    CASE OP_Arr_OP160P[Output_Page_num] OF
    700: OLine6:= "O140_LK_TST1 _SEL4(Q700.5)        ";
    701: OLine6:= "O140_LK_TST2 _SEL3(Q701.5)        ";
    702: OLine6:= "O140_LK_TST3 _SEL2(Q702.5)        ";
    703: OLine6:= "O140_LK_TST4 _SEL1(Q703.5)        ";
    704: OLine6:= "O140_LK_TST5 _STRT(Q704.5)        ";
    705: OLine6:= "O140_LK_TST6 _RST(Q705.5)         ";
    706: OLine6:= "O140_LK_TST6 _SEL7(Q706.5)        ";
    707: OLine6:= "O160_SAMPLE_PART_DOR_OPN(Q707.5) ";
    708: OLine6:= "O10A_DRUM_RST(Q708.5)             ";
    709: OLine6:= "O160_SPARE_Q709_5(Q709.5)         ";
   1340: OLine6:= "O130_LH_TOOL_CHO_LOCK(Q1340.5)";
   1341: OLine6:= "O140_TOOL1_CHO_LOCK(Q1341.5)";
   1342: OLine6:= "O140_TOOL2_CHO_LOCK(Q1342.5)";
   1343: OLine6:= "O140_TOOL3_CHO_LOCK(Q1343.5)";
   1350: OLine6:= "O160_SLIDE_CYL_FWD(Q1350.5)";
   1351: OLine6:= "O160_RH_PALLET_LOCK_CYL_LOCK(Q1351.5)";
   1352: OLine6:= "O160_SPARE_Q1352_5(Q1352.5)";
   1353: OLine6:= "O160_SPARE_Q1353_5(Q1353.5)";
    ELSE
      OLine6:= " ";	
    END_CASE
       Out_Visibility_6:=TRUE;
	
    CASE OP_Arr_OP160P[Output_Page_num] OF
	700:  Out_Lamp6:=O140_LK_TST1_SEL4_Q700_5;
	701:  Out_Lamp6:=O140_LK_TST2_SEL3_Q701_5;
	702:  Out_Lamp6:=O140_LK_TST3_SEL2_Q702_5;
	703:  Out_Lamp6:=O140_LK_TST4_SEL1_Q703_5;
	704:  Out_Lamp6:=O140_LK_TST5_STRT_Q704_5;
	705:  Out_Lamp6:=O140_LK_TST6_RST_Q705_5;
	706:  Out_Lamp6:=O140_LK_TST6_SEL7_Q706_5;
	707:  Out_Lamp6:=O160_SAMPLE_PART_DOOR_OPN_Q707_5;
	708:  Out_Lamp6:=O10A_DRUM_RST_Q708_5;
	709:  Out_Lamp6:=O160_SPARE_Q709_5;
	1340: Out_Lamp6:=O130_LH_TOOL_CHO_LOCK_Q1340_5;
	1341: Out_Lamp6:=O140_TOOL1_CHO_LOCK_Q1341_5;
	1342: Out_Lamp6:=O140_TOOL2_CHO_LOCK_Q1342_5;
	1343: Out_Lamp6:=O140_TOOL3_CHO_LOCK_Q1343_5;
	1350: Out_Lamp6:=O160_SLIDE_CYL_FWD_Q1350_5;
	1351: Out_Lamp6:=O160_RH_PALLET_LOCK_CYL_LOCK_Q1351_5;
	1352: Out_Lamp6:=O160_SPARE_Q1352_5;
	1353: Out_Lamp6:=O160_SPARE_Q1353_5;
   ELSE           
       Out_Visibility_6:=FALSE;
   END_CASE 
       
    CASE OP_Arr_OP160P[Output_Page_num] OF
    700: OLine7:= "O140_LK_TST1 _SEL5(Q700.6)    ";
    701: OLine7:= "O140_LK_TST2 _SEL4(Q701.6)    ";
    702: OLine7:= "O140_LK_TST3 _SEL3(Q702.6)    ";
    703: OLine7:= "O140_LK_TST4 _SEL2(Q703.6)    ";
    704: OLine7:= "O140_LK_TST5 _SEL1(Q704.6)    ";
    705: OLine7:= "O140_LK_TST6 _STRT(Q705.6)    ";
    706: OLine7:= "O150_VISN_LGHT_ON(Q706.6)     ";
    707: OLine7:= "O160_REJ_BIN_DOR_OPN(Q707.6) ";
    708: OLine7:= "O10A_DRUM_EXT_SPEED(Q708.6)   ";
    709: OLine7:= "O160_SPARE_Q709_6(Q709.6)     ";
   1340: OLine7:= "O130_RH_TOOL_CHO_UNLOCK(Q1340.6)";
   1341: OLine7:= "O140_WIPE1_CYL_REV(Q1341.6)";
   1342: OLine7:= "O140_WIPE2_CYL_REV(Q1342.6)";
   1343: OLine7:= "O140_WIPE3_CYL_REV(Q1343.6)";
   1350: OLine7:= "O160_SPARE_Q1350_6(Q1350.6)";
   1351: OLine7:= "O160_SPARE_Q1351_6(Q1351.6)";
   1352: OLine7:= "O160_SPARE_Q1352_6(Q1352.6)";
   1353: OLine7:= "O160_SPARE_Q1353_6(Q1353.6)";
    ELSE
      OLine7:= " ";	
    END_CASE
       Out_Visibility_7:=TRUE;
	
   CASE OP_Arr_OP160P[Output_Page_num] OF
	700:  Out_Lamp7:=O140_LK_TST1_SEL5_Q700_6;
	701:  Out_Lamp7:=O140_LK_TST2_SEL4_Q701_6;
	702:  Out_Lamp7:=O140_LK_TST3_SEL3_Q702_6;
	703:  Out_Lamp7:=O140_LK_TST4_SEL2_Q703_6;
	704:  Out_Lamp7:=O140_LK_TST5_SEL1_Q704_6;
	705:  Out_Lamp7:=O140_LK_TST6_STRT_Q705_6;
	706:  Out_Lamp7:=O150_VISN_LGHT_ON_Q706_6;
	707:  Out_Lamp7:=O160_REJ_BIN_DOOR_OPN_Q707_6;
	708:  Out_Lamp7:=O10A_DRUM_EXT_SPEED_Q708_6;
	709:  Out_Lamp7:=O160_SPARE_Q709_6;
	1340: Out_Lamp7:=O130_RH_TOOL_CHO_UNLOCK_Q1340_6;
	1341: Out_Lamp7:=O140_WIPE1_CYL_REV_Q1341_6;
	1342: Out_Lamp7:=O140_WIPE2_CYL_REV_Q1342_6;
	1343: Out_Lamp7:=O140_WIPE3_CYL_REV_Q1343_6;
	1350: Out_Lamp7:=O160_SPARE_Q1350_6;
	1351: Out_Lamp7:=O160_SPARE_Q1351_6;
	1352: Out_Lamp7:=O160_SPARE_Q1352_6;
	1353: Out_Lamp7:=O160_SPARE_Q1353_6;
   ELSE
       Out_Visibility_7:=FALSE;
   END_CASE 
    
    CASE OP_Arr_OP160P[Output_Page_num] OF
    700: OLine8:= "O140_LK_TST1_SEL6(Q700.7)";
    701: OLine8:= "O140_LK_TST2_SEL5(Q701.7)";
    702: OLine8:= "O140_LK_TST3_SEL4(Q702.7)";
    703: OLine8:= "O140_LK_TST4_SEL3(Q703.7)";
    704: OLine8:= "O140_LK_TST5_SEL2(Q704.7)";
    705: OLine8:= "O140_LK_TST6_SEL1(Q705.7)";
    706: OLine8:= "O150_BARLIGHT_OP1(Q706.7) ";
    707: OLine8:= "O160_SPARE(Q707.7)        ";
    708: OLine8:= "O160_SPARE_Q708_7(Q708.7) ";
    709: OLine8:= "O160_SPARE_Q709_7(Q709.7) ";
   1340: OLine8:= "O130_RH_TOOL_CHO_LOCK(Q1340.7)";
   1341: OLine8:= "O140_WIPE1_CYL_FWD(Q1341.7)";
   1342: OLine8:= "O140_WIPE2_CYL_FWD(Q1342.7)";
   1343: OLine8:= "O140_WIPE3_CYL_FWD(Q1343.7)";
   1350: OLine8:= "O160_SPARE_Q1350_7(Q1350.7)";
   1351: OLine8:= "O160_SPARE_Q1351_7(Q1351.7)";
   1352: OLine8:= "O160_SPARE_Q1352_7(Q1352.7)";
   1353: OLine8:= "O160_SPARE_Q1353_7(Q1353.7)";
    ELSE
      OLine8:= " ";	
    END_CASE	
       Out_Visibility_8:=TRUE;
   
   CASE OP_Arr_OP160P[Output_Page_num] OF
	700:  Out_Lamp8:=O140_LK_TST1_SEL6_Q700_7;
	701:  Out_Lamp8:=O140_LK_TST2_SEL5_Q701_7;
	702:  Out_Lamp8:=O140_LK_TST3_SEL4_Q702_7;
	703:  Out_Lamp8:=O140_LK_TST4_SEL3_Q703_7;
	704:  Out_Lamp8:=O140_LK_TST5_SEL2_Q704_7;
	705:  Out_Lamp8:=O140_LK_TST6_SEL1_Q705_7;
	706:  Out_Lamp8:=O150_BARLIGHT_OP1_Q706_7;
	707:  Out_Lamp8:=O160_SPARE_Q707_7;
	708:  Out_Lamp8:=O160_SPARE_Q708_7;
	709:  Out_Lamp8:=O160_SPARE_Q709_7;
	1340: Out_Lamp8:=O130_RH_TOOL_CHO_LOCK_Q1340_7;
	1341: Out_Lamp8:=O140_WIPE1_CYL_FWD_Q1341_7;
	1342: Out_Lamp8:=O140_WIPE2_CYL_FWD_Q1342_7;
	1343: Out_Lamp8:=O140_WIPE3_CYL_FWD_Q1343_7;
	1350: Out_Lamp8:=O160_SPARE_Q1350_7;
	1351: Out_Lamp8:=O160_SPARE_Q1351_7;
	1352: Out_Lamp8:=O160_SPARE_Q1352_7;
	1353: Out_Lamp8:=O160_SPARE_Q1353_7;
   ELSE
       Out_Visibility_8:=FALSE;	
   END_CASE 
  
 4: CASE IP_Arr_OP10A[Input_Page_num] OF
      100:Line1:="I10A_HPR_UNIT_ALRM(I100.0)    ";
      101:Line1:="I10A_HPR_DOOR_SELCTN(I101.0)  ";
      102:Line1:="I10A_LNR_TRK1_CHO_MOD1(I102.0)";
      103:Line1:="I10A_SPARE_I103_0(I103.0)     ";
      ELSE
      	Line1:= " ";
      END_CASE
      
      CASE IP_Arr_OP10A[Input_Page_num] OF
      100:Line2:="I10A_SPARE_I100.1(I100.1)      ";
      101:Line2:="I10A_SPARE_I101.1(I101.1)      ";
      102:Line2:="I10A_LNR_TRK1_CHO_MOD2(I102.1) ";
      103:Line2:="I10A_SPARE_I103_1(I103.1)      ";
      ELSE
      	Line2 := " ";
      END_CASE
      
      CASE IP_Arr_OP10A[Input_Page_num] OF
      100:Line3:="I10A_HPR_LOW_LVL_SEN(I100.2)   ";
      101:Line3:="I10A_BDY_BOWL_LOW_LVL(I101.2)  ";
      102:Line3:="I10A_LNR_TRK2_CHO_MOD1(I102.2) ";
      103:Line3:="I10A_SPARE_I103_2(I103.2)      ";
      ELSE
      	Line3 := " ";
      END_CASE
      
      CASE IP_Arr_OP10A[Input_Page_num] OF
      100:Line4:="I10A_HPR_SOL_DOOR_SW_FB(I100.3)";
      101:Line4:="I10A_BDY_BWL_RUN(I101.3)       ";
      102:Line4:="I10A_LNR_TRK2_CHO_MOD2(I102.3) ";
      103:Line4:="I10A_SPARE_I103_3(I103.3)      ";
      ELSE
      	Line4 := " ";
      END_CASE
      
      CASE IP_Arr_OP10A[Input_Page_num] OF
      100:Line5:="I10A_HPR_OFF_ON(I100.4)";
      101:Line5:="I10A_BDY_LNR1_RUN(I101.4)";
      102:Line5:="I10A_SPARE_I102_4(I102.4)";
      103:Line5:="I10A_SPARE_I103_4(I103.4)";
      ELSE
      	Line5:= " ";
      END_CASE
      
      CASE IP_Arr_OP10A[Input_Page_num] OF
      100:Line6:="I10A_BDY_BOWL_OFF_ON(I100.5)  ";
      101:Line6:="I10A_BDY_LNR2_RUN(I101.5)     ";
      102:Line6:="I10A_SPARE_I102_5(I102.5)";
      103:Line6:="I10A_SPARE_I103_5(I103.5)     ";
      ELSE
      	Line6 := " ";
      END_CASE
      
      CASE IP_Arr_OP10A[Input_Page_num] OF
      100:Line7:="I10A_BDY_LNR1_OFF_ON(I100.6)     ";
      101:Line7:="I10A_BDY_LNR_FEED1_OVRFLW(I101.6)";
      102:Line7:="I10A_LH_BDY_CONT_FB(I102.6)      ";
      103:Line7:="I10A_SPARE_I103_6(I103.6)        ";
      ELSE
      	Line7 := " ";
      END_CASE
      
      CASE IP_Arr_OP10A[Input_Page_num] OF
      100:Line8:="I10A_BDY_LNR2_OFF_ON(I100.7)     ";
      101:Line8:="I10A_BDY_LNR_FEED2_OVRFLW(I101.7)";
      102:Line8:="I10A_RH_BDY_CONT_FB(I102.7)      ";
      103:Line8:="I10A_SPARE_I103_7(I103.7)        ";
      ELSE
      	Line8 := " ";
      END_CASE
	 	Visibility_1:=TRUE;
   
   CASE IP_Arr_OP10A[Input_Page_num] OF
	100: Lamp1:=I10A_HPR_UNIT_ALRM_I100_0 ;
	101: Lamp1:=I10A_HPR_DOOR_SELCTN_I101_0 ;
	102: Lamp1:=I10A_LNR_TRK1_CHO_MOD1_I102_0 ;
	103: Lamp1:=I10A_SPARE_I103_0;
   ELSE
       Visibility_1:=FALSE;	
   END_CASE
   
   Visibility_2:=TRUE;
   
   CASE IP_Arr_OP10A[Input_Page_num] OF
	100: Lamp2:=I10A_SPARE_I100_1 ;
	101: Lamp2:=I10A_SPARE_I101_1;
	102: Lamp2:=I10A_LNR_TRK1_CHO_MOD2_I102_1 ;
	103: Lamp2:=I10A_SPARE_I103_1;
   ELSE
       Visibility_2:=FALSE;	
   END_CASE
   
   
    Visibility_3:=TRUE;
   
   CASE IP_Arr_OP10A[Input_Page_num] OF
	100: Lamp3:=I10A_HPR_LOW_LVL_SEN_I100_2 ;
	101: Lamp3:=I10A_BDY_BOWL_LOW_LVL_I101_2 ;
	102: Lamp3:=I10A_LNR_TRK2_CHO_MOD1_I102_2 ;
	103: Lamp3:=I10A_SPARE_I103_2;
   ELSE
       Visibility_3:=FALSE;	
   END_CASE
   
   
    Visibility_4:=TRUE;
   
   CASE IP_Arr_OP10A[Input_Page_num] OF
	100: Lamp4:=I10A_HPR_SOL_DOOR_SW_FB_I100_3 ;
	101: Lamp4:=I10A_BDY_BWL_RUN_I101_3 ;
	102: Lamp4:=I10A_LNR_TRK2_CHO_MOD2_I102_3 ;
	103: Lamp4:=I10A_SPARE_I103_3;
   ELSE
       Visibility_4:=FALSE;	
   END_CASE
   
   
    
    Visibility_5:=TRUE;
   
   CASE IP_Arr_OP10A[Input_Page_num] OF
	100: Lamp5:=I10A_HPR_OFF_ON_I100_4 ;
	101: Lamp5:=I10A_BDY_LNR1_RUN_I101_4 ;
	102: Lamp5:=I10A_SPARE_I102_4 ;
	103: Lamp5:=I10A_SPARE_I103_4;
   ELSE
       Visibility_5:=FALSE;	
   END_CASE
   
    
    Visibility_6:=TRUE;
   
   CASE IP_Arr_OP10A[Input_Page_num] OF
	100: Lamp6:=I10A_BDY_BOWL_OFF_ON_I100_5 ;
	101: Lamp6:=I10A_BDY_LNR2_RUN_I101_5 ;
	102: Lamp6:=I10A_SPARE_I102_5 ;
	103: Lamp6:=I10A_SPARE_I103_5;
   ELSE
       Visibility_6:=FALSE;	
   END_CASE
   
   
      
    Visibility_7:=TRUE;
   
   CASE IP_Arr_OP10A[Input_Page_num] OF
	100: Lamp7:=I10A_BDY_LNR1_OFF_ON_I100_6 ;
	101: Lamp7:=I10A_BDY_LNR_FEED1_OVRFLW_I101_6 ;
	102: Lamp7:=I10A_LH_BDY_CONT_FB_I102_6;
	103: Lamp7:=I10A_SPARE_I103_6;
   ELSE
       Visibility_7:=FALSE;	
   END_CASE


 	Visibility_8:=TRUE;
   
   CASE IP_Arr_OP10A[Input_Page_num] OF
	100: Lamp8:=I10A_BDY_LNR2_OFF_ON_I100_7 ;
	101: Lamp8:=I10A_BDY_LNR_FEED2_OVRFLW_I101_7 ;
	102: Lamp8:=I10A_RH_BDY_CONT_FB_I102_7 ;
	103: Lamp8:=I10A_SPARE_I103_7;
   ELSE
       Visibility_8:=FALSE;	
   END_CASE

	
	 CASE OP_Arr_OP10A[Output_Page_num] OF
     100:OLine1:="O10A_HPR_MTR_FWD(Q100.0)  ";
     101:OLine1:="O10A_BDY_BOWL_ON(Q101.0)  ";
     102:OLine1:="O10A_SPARE_Q102_0(Q102.0) ";
     103:OLine1:="O10A_SPARE_Q103_0(Q103.0) ";
     ELSE
     	OLine1:= " ";
     END_CASE
     
     CASE OP_Arr_OP10A[Output_Page_num] OF
     100:OLine2:="O10A_HPR_RST(Q100.1)         ";
     101:OLine2:="O10A_BDY_LNR_FEED1_ON(Q101.1)";
     102:OLine2:="O10A_SPARE_Q102_1(Q102.1)    ";
     103:OLine2:="O10A_SPARE_Q103_1(Q103.1)    ";
     ELSE
     	OLine2:= " ";
     END_CASE
     
     CASE OP_Arr_OP10A[Output_Page_num] OF
     100:OLine3:="O10A_EXT_SPEED(Q100.2)       ";
     101:OLine3:="O10A_BDY_LNR_FEED2_ON(Q101.2)";
     102:OLine3:="O10A_SPARE_Q102_2(Q102.2)    ";
     103:OLine3:="O10A_SPARE_Q103_2(Q103.2)    ";
     ELSE
     	OLine3:= " ";
     END_CASE
     
     CASE OP_Arr_OP10A[Output_Page_num] OF
     100:OLine4:="O10A_SPARE_Q100.3(Q100.3)      ";
     101:OLine4:="O10A_BDY_LNR1_AIR_PURGE(Q101.3)";
     102:OLine4:="O10A_SPARE_Q102_3(Q102.3)      ";
     103:OLine4:="O10A_SPARE_Q103_3(Q103.3)      ";
     ELSE
     	OLine4:= " ";
     END_CASE
     
     CASE OP_Arr_OP10A[Output_Page_num] OF
     100:OLine5:="O10A_HPR_DOOR_SELCTN_IND(Q100.4)";
   //101:OLine5:="O10A_BDY_LNR2_AIRPURGE(Q101.4)";
     102:OLine5:="O10A_SPARE_Q102_4(Q102.4)";
     103:OLine5:="O10A_SPARE_Q103_4(Q103.4)";
     ELSE
     	OLine5:= " ";
     END_CASE
     
     CASE OP_Arr_OP10A[Output_Page_num] OF
     100:OLine6:="O10A_HPR_TWR_LMP_RED(Q100.5)";
     101:OLine6:="O10A_HPR_DOOR_OPN(Q101.5)   ";
     102:OLine6:="O10A_SPARE_Q102_5(Q102.5)   ";
     103:OLine6:="O10A_SPARE_Q103_5(Q103.5)   ";
     ELSE
     	OLine6:= " ";
     END_CASE
     
     CASE OP_Arr_OP10A[Output_Page_num] OF
     100:OLine7:="O10A_HPR_TWR_LMP_GREEN(Q100.6)";
     101:OLine7:="O10A_SPARE_Q101_6(Q101.6)     ";
     102:OLine7:="O10A_SPARE_Q102_6(Q102.6)     ";
     103:OLine7:="O10A_SPARE_Q103_6(Q103.6)     ";
     ELSE
     	OLine7:= " ";
     END_CASE
     
     CASE OP_Arr_OP10A[Output_Page_num] OF
     100:OLine8:="O10A_SPARE_Q100_7(Q100.7)";
     101:OLine8:="O10A_SPARE_Q101_7(Q101.7)";
     102:OLine8:="O10A_SPARE_Q102_7(Q102.7)";
     103:OLine8:="O10A_SPARE_Q103_7(Q103.7)";
     ELSE
     	OLine8:= " ";
     END_CASE
	  Out_Visibility_1:=TRUE;

    CASE OP_Arr_OP10A[Output_Page_num] OF
	100:  Out_Lamp1:=O10A_HPR_MTR_FWD_Q100_0;
	101:  Out_Lamp1:=O10A_BDY_BOWL_ON_Q101_0;
	102:  Out_Lamp1:=O10A_SPARE_Q102_0;
	103:  Out_Lamp1:=O10A_SPARE_Q103_0;
   ELSE
       Out_Visibility_1:=FALSE;	
   END_CASE
   
    Out_Visibility_2:=TRUE;
   
   CASE OP_Arr_OP10A[Output_Page_num] OF
	100:  Out_Lamp2:=O10A_HPR_RST_Q100_1;
	101:  Out_Lamp2:=O10A_BDY_LNR_FEED1_ON_Q101_1;
	102:  Out_Lamp2:=O10A_SPARE_Q102_1;
	103:  Out_Lamp2:=O10A_SPARE_Q103_1;
   ELSE
       Out_Visibility_2:=FALSE;	
   END_CASE 
   
    Out_Visibility_3:=TRUE;
	
   CASE OP_Arr_OP10A[Output_Page_num] OF
	100:  Out_Lamp3:=O10A_EXT_SPEED_Q100_2; 
	101:  Out_Lamp3:=O10A_BDY_LNR_FEED2_ON_Q101_2; 
	102:  Out_Lamp3:=O10A_SPARE_Q102_2; 
	103:  Out_Lamp3:=O10A_SPARE_Q103_2; 
   ELSE
       Out_Visibility_3:=FALSE;
   END_CASE 
   
    Out_Visibility_4:=TRUE;
   
   CASE OP_Arr_OP10A[Output_Page_num] OF
	100:  Out_Lamp4:=O10A_SPARE_Q100_3; 
	101:  Out_Lamp4:=O10A_BDY_LNR1_AIR_PURGE_Q101_3; 
	102:  Out_Lamp4:=O10A_SPARE_Q102_3; 
	103:  Out_Lamp4:=O10A_SPARE_Q103_3;  
   ELSE
       Out_Visibility_4:=FALSE;
   END_CASE 
   
    Out_Visibility_5:=TRUE;
	
    CASE OP_Arr_OP10A[Output_Page_num] OF
	100:  Out_Lamp5:=O10A_HPR_DOOR_SELCTN_IND_Q100_4; 
	//101:  Out_Lamp5:=O10A_BDY_LNR2_AIR_PURGE_Q101_4; 
	102:  Out_Lamp5:=O10A_SPARE_Q102_4; 
	103:  Out_Lamp5:=O10A_SPARE_Q103_4; 	 
   ELSE
       Out_Visibility_5:=FALSE;
   END_CASE 
   
    Out_Visibility_6:=TRUE;
	
   CASE OP_Arr_OP10A[Output_Page_num] OF
	100:  Out_Lamp6:=O10A_HPR_TWR_LMP_RED_Q100_5; 
	101:  Out_Lamp6:=O10A_HPR_DOOR_OPN_Q101_5; 
	102:  Out_Lamp6:=O10A_SPARE_Q102_5; 
	103:  Out_Lamp6:=O10A_SPARE_Q103_5; 
   ELSE           
       Out_Visibility_6:=FALSE;
   END_CASE 
    
	Out_Visibility_7:=TRUE;
	
   CASE OP_Arr_OP10A[Output_Page_num] OF
	100:  Out_Lamp7:=O10A_HPR_TWR_LMP_GREEN_Q100_6; 
	101:  Out_Lamp7:=O10A_SPARE_Q101_6; 
	102:  Out_Lamp7:=O10A_SPARE_Q102_6; 
	103:  Out_Lamp7:=O10A_SPARE_Q103_6;  
   ELSE 
       Out_Visibility_7:=FALSE;
   END_CASE 
   
    Out_Visibility_8:=TRUE;
   
   CASE OP_Arr_OP10A[Output_Page_num] OF
	100:  Out_Lamp8:=O10A_SPARE_Q100_7;  
	101:  Out_Lamp8:=O10A_SPARE_Q101_7;  
	102:  Out_Lamp8:=O10A_SPARE_Q102_7;  
	103:  Out_Lamp8:=O10A_SPARE_Q103_7;   
   ELSE
       Out_Visibility_8:=FALSE;	
   END_CASE
	 
 5: CASE IP_Arr_OP10B[Input_Page_num] OF
    200: Line1:= "I10B_HPR_UNIT_ALRM(I200.0)     ";
    201: Line1:= "I10B_HPR_DOOR_SELCTN(I201.0)   ";
    202: Line1:= "I10B_LNR_TRK1_CHO_MOD1(I202.0) ";
    203: Line1:= "I10B_SPARE_I203_0(I203.0)      ";
    ELSE
    	Line1 := " ";
    END_CASE
    
    CASE IP_Arr_OP10B[Input_Page_num] OF
    200: Line2:= "I10B_SPARE_I200_1(I200.1)     ";
    201: Line2:= "I10B_SPARE_I201_1(I201.1)     ";
    202: Line2:= "I10B_LNR_TRK1_CHO_MOD2(I202.1)";
    203: Line2:= "I10B_SPARE_I203_1(I203.1)     ";
    ELSE
    	Line2 := " ";
    END_CASE
    
    CASE IP_Arr_OP10B[Input_Page_num] OF
    200: Line3:= "I10B_HPR_LOW_LVL_SEN(I200.2)   ";
    201: Line3:= "I10B_BDY_BOWL_LOW_LVL(I201.2)  ";
    202: Line3:= "I10B_LNR_TRK2_CHO_MOD1(I202.2) ";
    203: Line3:= "I10B_SPARE_I203_2(I203.2)      ";
    ELSE
    	Line3 := " ";
    END_CASE
    
    CASE IP_Arr_OP10B[Input_Page_num] OF
    200: Line4:= "I10B_HPR_SOL_DOOR_SW_FB(I200.3)";
    201: Line4:= "I10B_BDY_BWL_RUN(I201.3)       ";
    202: Line4:= "I10B_LNR_TRK2_CHO_MOD2(I202.3) ";
    203: Line4:= "I10B_SPARE_I203_3(I203.3)      ";
    ELSE
    	Line4 := " ";
    END_CASE
    
    CASE IP_Arr_OP10B[Input_Page_num] OF
    200: Line5:= "I10B_HPR_OFF_ON(I200.4)       ";
    201: Line5:= "I10B_BDY_LNR1_RUN(I201.4)     ";
    202: Line5:= "I10B_SPARE_I202_4(I202.4)";
    203: Line5:= "I10B_SPARE_I203_4(I203.4)     ";
    ELSE
    	Line5 := " ";
    END_CASE
    
    CASE IP_Arr_OP10B[Input_Page_num] OF
    200: Line6:= "I10B_BDY_BOWL_OFF_ON(I200.5)   ";
    201: Line6:= "I10B_BDY_LNR2_RUN(I201.5)      ";
    202: Line6:= "I10B_SPARE_I202_5(I202.5) ";
    203: Line6:= "I10B_SPARE_I203_5(I203.5)      ";
    ELSE
    	Line6 := " ";
    END_CASE
    
    CASE IP_Arr_OP10B[Input_Page_num] OF
    200: Line7:= "I10B_BDY_LNR1_OFF_ON(I200.6)      ";
    201: Line7:= "I10B_BDY_LNR_FEED1_OVRFLW(I201.6) ";
    202: Line7:= "I10B_SPARE_I202_6(I202.6)         ";
    203: Line7:= "I10B_SPARE_I203_6(I203.6)         ";
    ELSE
    	Line7 := " ";
    END_CASE
    
    CASE IP_Arr_OP10B[Input_Page_num] OF
    200: Line8:= "I10B_BDY_LNR2_OFF_ON(I200.7)     ";
    201: Line8:= "I10B_BDY_LNR_FEED2_OVRFLW(I201.7)";
    202: Line8:= "I10B_SPARE_I202_7(I202.7)        ";
    203: Line8:= "I10B_SPARE_I203_7(I203.7)        ";
    ELSE
    	Line8 := " ";
    END_CASE
	  Visibility_1:=TRUE;
   
   CASE IP_Arr_OP10B[Input_Page_num] OF
	200: Lamp1:=I10B_HPR_UNIT_ALRM_I200_0 ;
	201: Lamp1:=I10B_HPR_DOOR_SELCTN_I201_0 ;
	202: Lamp1:=I10B_LNR_TRK1_CHO_MOD1_I202_0 ;
	203: Lamp1:=I10B_SPARE_I203_0;
   ELSE
       Visibility_1:=FALSE;	
   END_CASE
   
   
   Visibility_2:=TRUE;
   
   CASE IP_Arr_OP10B[Input_Page_num] OF
	200: Lamp2:=I10B_SPARE_I200_1 ;
	201: Lamp2:=I10B_SPARE_I201_1 ;
	202: Lamp2:=I10B_LNR_TRK1_CHO_MOD2_I202_1 ;
	203: Lamp2:=I10B_SPARE_I203_1;
   ELSE
       Visibility_2:=FALSE;	
   END_CASE
   
   
    Visibility_3:=TRUE;
   
   CASE IP_Arr_OP10B[Input_Page_num] OF
	200: Lamp3:=I10B_HPR_LOW_LVL_SEN_I200_2 ;
	201: Lamp3:=I10B_BDY_BOWL_LOW_LVL_I201_2 ; 
	202: Lamp3:=I10B_LNR_TRK2_CHO_MOD1_I202_2 ;
	203: Lamp3:=I10B_SPARE_I203_2 ;
   ELSE
       Visibility_3:=FALSE;	
   END_CASE
   
   
    Visibility_4:=TRUE;
   
   CASE IP_Arr_OP10B[Input_Page_num] OF
	200: Lamp4:=I10B_HPR_SOL_DOOR_SW_FB_I200_3 ;
	201: Lamp4:=I10B_BDY_BWL_RUN_I201_3 ; 
	202: Lamp4:=I10B_LNR_TRK2_CHO_MOD2_I202_3 ;
	203: Lamp4:=I10B_SPARE_I203_3 ;
   ELSE
       Visibility_4:=FALSE;	
   END_CASE
   
   
    Visibility_5:=TRUE;
   
   CASE IP_Arr_OP10B[Input_Page_num] OF
	200: Lamp5:=I10B_HPR_OFF_ON_I200_4 ;
	201: Lamp5:=I10B_BDY_LNR1_RUN_I201_4 ;
	202: Lamp5:=I10B_SPARE_I202_4 ;
	203: Lamp5:=I10B_SPARE_I203_4;
   ELSE
       Visibility_5:=FALSE;	
   END_CASE
   
    
    Visibility_6:=TRUE;
   
   CASE IP_Arr_OP10B[Input_Page_num] OF
	200: Lamp6:=I10B_BDY_BOWL_OFF_ON_I200_5 ;
	201: Lamp6:=I10B_BDY_LNR2_RUN_I201_5 ;
	202: Lamp6:=I10B_SPARE_I202_5 ;
	203: Lamp6:=I10B_SPARE_I203_5 ;
   ELSE
       Visibility_6:=FALSE;	
   END_CASE
   
      
    Visibility_7:=TRUE;
   
   CASE IP_Arr_OP10B[Input_Page_num] OF
	200: Lamp7:=I10B_BDY_LNR1_OFF_ON_I200_6 ;
	201: Lamp7:=I10B_BDY_LNR_FEED1_OVRFLW_I201_6 ;
	202: Lamp7:=I10B_SPARE_I202_6 ;
	203: Lamp7:=I10B_SPARE_I203_6;
   ELSE
       Visibility_7:=FALSE;	
   END_CASE


    Visibility_8:=TRUE;
   
   CASE IP_Arr_OP10B[Input_Page_num] OF
	200: Lamp8:=I10B_BDY_LNR2_OFF_ON_I200_7 ;
	201: Lamp8:=I10B_BDY_LNR_FEED2_OVRFLW_I201_7 ;
	202: Lamp8:=I10B_SPARE_I202_7 ;
	203: Lamp8:=I10B_SPARE_I203_7;
   ELSE
       Visibility_8:=FALSE;	
   END_CASE


  CASE OP_Arr_OP10B_JB[Output_Page_num] OF	
  200: OLine1:= " O10B_HPR_MTR_FWD(Q200.0) ";
  201: OLine1:= " O10B_BDY_BOWL_ON(Q201.0) ";
  202: OLine1:= " O10B_SPARE_Q202_0(Q202.0)";
  203: OLine1:= " O10B_SPARE_Q203_0(Q203.0)";
  ELSE
      OLine1 := " ";
  END_CASE
  
  CASE OP_Arr_OP10B_JB[Output_Page_num] OF
  200: OLine2:= "O10B_HPR_RST(Q200.1)         ";
  201: OLine2:= "O10B_BDY_LNR_FEED1_ON(Q201.1)";
  202: OLine2:= "O10B_SPARE_Q202_1(Q202.1)    ";
  203: OLine2:= "O10B_SPARE_Q203_1(Q203.1)    ";
  ELSE
    OLine2 := " ";
  END_CASE
  
  CASE OP_Arr_OP10B_JB[Output_Page_num] OF
  200: OLine3:= "O10B_EXT_SPEED(Q200.2)       ";
  201: OLine3:= "O10B_BDY_LNR_FEED2_ON(Q201.2)";
  202: OLine3:= "O10B_SPARE_Q202_2(Q202.2)    ";
  203: OLine3:= "O10B_SPARE_Q2032_(Q203.2)    ";
  ELSE
    OLine3 := " ";
  END_CASE
  
  CASE OP_Arr_OP10B_JB[Output_Page_num] OF
  200: OLine4:= "O10B_SPARE_Q200.3(Q200.3)      ";
  201: OLine4:= "O10B_BDY_LNR1_AIR_PURGE(Q201.3)";
  202: OLine4:= "O10B_SPARE_Q202_3(Q202.3)      ";
  203: OLine4:= "O10B_SPARE_Q203_3(Q203.3)      ";
  ELSE
    OLine4 := " ";
  END_CASE
  
  CASE OP_Arr_OP10B_JB[Output_Page_num] OF
  200: OLine5:= "O10B_HPR_DOOR_SELCTN_IND(Q200.4)";
  //201: OLine5:= "O10B_BDY_LNR2_AIR_PURGE(Q201.4) ";
  202: OLine5:= "O10B_SPARE_Q202_4(Q202.4)       ";
  203: OLine5:= "O10B_SPARE_Q203_4(Q203.4)       ";
  ELSE
     OLine5 := " ";
  END_CASE
  
  CASE OP_Arr_OP10B_JB[Output_Page_num] OF
  200: OLine6:= "O10B_HPR_TWR_LMP_RED(Q200.5)";
  201: OLine6:= "O10B_HPR_DOOR_OPN(Q201.5)   ";
  202: OLine6:= "O10B_SPARE_Q202_5(Q202.5)   ";
  203: OLine6:= "O10B_SPARE_Q203_5(Q203.5)   ";
  ELSE
     OLine6 := " ";
  END_CASE
  
  CASE OP_Arr_OP10B_JB[Output_Page_num] OF
  200: OLine7:= "O10B_HPR_TWR_LMP_GREEN(Q200.6)";
  201: OLine7:= "O10B_SPARE_Q201_6(Q201.6)     ";
  202: OLine7:= "O10B_SPARE_Q202_6(Q202.6)     ";
  203: OLine7:= "O10B_SPARE_Q203_6(Q203.6)     ";
  ELSE
      OLine7 := " ";
  END_CASE
  
  CASE OP_Arr_OP10B_JB[Output_Page_num] OF	 
  200: OLine8:= "O10B_SPARE_Q200_7(Q200.7)";
  201: OLine8:= "O10B_SPARE_Q201_7(Q201.7)";
  202: OLine8:= "O10B_SPARE_Q202_7(Q202.7)";
  203: OLine8:= "O10B_SPARE_Q203_7(Q203.7)";
  ELSE
      OLine8 := " ";
  END_CASE	

    Out_Visibility_1:=TRUE;

   CASE OP_Arr_OP10B_JB[Output_Page_num] OF
	200:  Out_Lamp1:=O10B_HPR_MTR_FWD_Q200_0;
	201:  Out_Lamp1:=O10B_BDY_BOWL_ON_Q201_0;
	202:  Out_Lamp1:=O10B_SPARE_Q202_0;
	203:  Out_Lamp1:=O10B_SPARE_Q203_0;
   ELSE
       Out_Visibility_1:=FALSE;	
   END_CASE
   
    Out_Visibility_2:=TRUE;
   
   CASE OP_Arr_OP10B_JB[Output_Page_num] OF
	200:  Out_Lamp2:=O10B_HPR_RST_Q200_1;
	201:  Out_Lamp2:=O10B_BDY_LNR_FEED1_ON_Q201_1;
	202:  Out_Lamp2:=O10B_SPARE_Q202_1;
	203:  Out_Lamp2:=O10B_SPARE_Q203_1;
   ELSE
       Out_Visibility_2:=FALSE;	
   END_CASE 
   
    Out_Visibility_3:=TRUE;
	
   CASE OP_Arr_OP10B_JB[Output_Page_num] OF
	200:  Out_Lamp3:=O10B_EXT_SPEED_Q200_2; 
	201:  Out_Lamp3:=O10B_BDY_LNR_FEED2_ON_Q201_2; 
	202:  Out_Lamp3:=O10B_SPARE_Q202_2; 
	203:  Out_Lamp3:=O10B_SPARE_Q203_2; 
   ELSE
       Out_Visibility_3:=FALSE;
   END_CASE 
   
    Out_Visibility_4:=TRUE;
   
   CASE OP_Arr_OP10B_JB[Output_Page_num] OF
	200:  Out_Lamp4:=O10B_SPARE_Q200_3; 
	201:  Out_Lamp4:=O10B_BDY_LNR1_AIR_PURGE_Q201_3; 
	202:  Out_Lamp4:=O10B_SPARE_Q202_3; 
	203:  Out_Lamp4:=O10B_SPARE_Q203_3;  
   ELSE
       Out_Visibility_4:=FALSE;
   END_CASE 
   
    Out_Visibility_5:=TRUE;
	
    CASE OP_Arr_OP10B_JB[Output_Page_num] OF
	200:  Out_Lamp5:=O10B_HPR_DOOR_SELCTN_IND_Q200_4; 
	201:  Out_Lamp5:=O10B_BDY_LNR2_AIR_PURGE_Q201_4 ; 
	202:  Out_Lamp5:=O10B_SPARE_Q202_4; 
	203:  Out_Lamp5:=O10B_SPARE_Q203_4; 	 
   ELSE
       Out_Visibility_5:=FALSE;
   END_CASE 
   
    Out_Visibility_6:=TRUE;
	
   CASE OP_Arr_OP10B_JB[Output_Page_num] OF
	200:  Out_Lamp6:=O10B_HPR_TWR_LMP_RED_Q200_5; 
	201:  Out_Lamp6:=O10B_HPR_DOOR_OPN_Q201_5; 
	202:  Out_Lamp6:=O10B_SPARE_Q202_5; 
	203:  Out_Lamp6:=O10B_SPARE_Q203_5; 
   ELSE           
       Out_Visibility_6:=FALSE;
   END_CASE 
    
	Out_Visibility_7:=TRUE;
	
   CASE OP_Arr_OP10B_JB[Output_Page_num] OF
	200:  Out_Lamp7:=O10B_HPR_TWR_LMP_GREEN_Q200_6; 
	201:  Out_Lamp7:=O10B_SPARE_Q201_6; 
	202:  Out_Lamp7:=O10B_SPARE_Q202_6; 
	203:  Out_Lamp7:=O10B_SPARE_Q203_6;  
   ELSE 
       Out_Visibility_7:=FALSE;
   END_CASE 
   
    Out_Visibility_8:=TRUE;
   
   CASE OP_Arr_OP10B_JB[Output_Page_num] OF
	200:  Out_Lamp8:=O10B_SPARE_Q200_7;  
	201:  Out_Lamp8:=O10B_SPARE_Q201_7;  
	202:  Out_Lamp8:=O10B_SPARE_Q202_7;  
	203:  Out_Lamp8:=O10B_SPARE_Q203_7;   
   ELSE
       Out_Visibility_8:=FALSE;	
   END_CASE 
 6: CASE IP_Arr_OP90JB[Input_Page_num] OF
    500: Line1:=" I90_SPARE_I500_0(I500.0)       ";
    501: Line1:=" I90_CONV1_FWD(I501.0)          ";
    502: Line1:=" I90_CONV1_TRK3_CHO_MOD2(I502.0)";
    503: Line1:=" I90_CONV2_REV(I503.0)          ";
    504: Line1:=" I90_CONV2_TRK3_CHO_MOD1(I504.0)";
    505: Line1:=" I90_SPARE_I505_0(I505.0)       ";
    else
     Line1:=" ";
    end_case 
    
    CASE IP_Arr_OP90JB[Input_Page_num] OF
    500: Line2:="I90_HPR1_LOW_LVL_FB(I500.1)        ";
    501: Line2:="I90_VBF1_CONV1_TRK1_OVERFLW(I501.1)";
    502: Line2:="I90_SPARE_I502_1(I502.1)           ";
    503: Line2:="I90_CONV2_FWD(I503.1)              ";
    504: Line2:="I90_CONV2_TRK3_CHO_MOD2(I504.1)    ";
    505: Line2:="I90_SPARE_I505_1(I505.1)           ";
    else
     Line2:=" ";
    end_case 
    
    CASE IP_Arr_OP90JB[Input_Page_num] OF
    500: Line3:="I90_HPR1_SOL_DOOR_SW_FB(I500.2)    ";
    501: Line3:="I90_VBF1_CONV1_TRK2_OVERFLW(I501.2)";
    502: Line3:="I90_HPR2_LOW_LVL_FB(I502.2)        ";
    503: Line3:="I90_VBF1_CONV2_TRK1_OVERFLW(I503.2)";
    504: Line3:="I90_VBF1_CONV_TRK_OVERFLW_2(I504.2)";
    505: Line3:="I90_SPARE_I505_2(I505.2)           ";
    else
     Line3:=" ";
    end_case 
    
    CASE IP_Arr_OP90JB[Input_Page_num] OF
    500: Line4:="I90_BOWL1_RDY(I500.3)              ";
    501: Line4:="I90_CONV1_TRK1_CHO_MOD1(I501.3)    ";
    502: Line4:="I90_HPR2_SOL_DOOR_SW_FB(I502.3)    ";
    503: Line4:="I90_VBF1_CONV2_TRK2_OVERFLW(I503.3)";
    504: Line4:="I90_VBF2_CONV_TRK_OVERFLW_2(I504.3)";
    505: Line4:="I90_SPARE_I505_3(I505.3)           ";
    else
     Line4:=" ";
    end_case 
    
    CASE IP_Arr_OP90JB[Input_Page_num] OF
    500: Line5:="I90_BOWL1_LOW_LVL(I500.4)      ";
    501: Line5:="I90_CONV1_TRK1_CHO_MOD2(I501.4)";
    502: Line5:="I90_BOWL2_RDY(I502.4)          ";
    503: Line5:="I90_CONV2_TRK1_CHO_MOD1(I503.4)";
    504: Line5:="I90_SPARE_I504_4(I504.4)       ";
    505: Line5:="I90_SPARE_I505_4(I505.4)       ";
    else
     Line5:=" ";
    end_case 
    
    CASE IP_Arr_OP90JB[Input_Page_num] OF
    500: Line6:="I90_BOWL1_OFF_ON(I500.5)        ";
    501: Line6:="I90_CONV1_TRK2_CHO_MOD1(I501.5) ";
    502: Line6:="I90_BOWL2_LOW_LVL(I502.5)       ";
    503: Line6:="I90_CONV2_TRK1_CHO_MOD2(I503.5) ";
    504: Line6:="I90_SPARE_I504_5(I504.5)        ";
    505: Line6:="I90_SPARE_I505_5(I505.5)        ";
    else
     Line6:=" ";
    end_case 
    
    CASE IP_Arr_OP90JB[Input_Page_num] OF
    500: Line7:="I90_HPR1_OFF_ON(I500.6)        ";
    501: Line7:="I90_CONV1_TRK2_CHO_MOD2(I501.6)";
    502: Line7:="I90_BOWL2_OFF_ON(I502.6)       ";
    503: Line7:="I90_CONV2_TRK2_CHO_MOD1(I503.6)";
    504: Line7:="I90_SPARE_I504_6(I504.6)       ";
    505: Line7:="I90_SPARE_I505_6(I505.6)       ";
    else
     Line7:=" ";
    end_case 
    
    CASE IP_Arr_OP90JB[Input_Page_num] OF
    500: Line8:="I90_CONV1_REV(I500.7)           ";
    501: Line8:="I90_CONV1_TRK3_CHO_MOD1(I501.7) ";
    502: Line8:="I90_HPR2_OFF_ON(I502.7)         ";
    503: Line8:="I90_CONV2_TRK2_CHO_MOD2(I503.7) ";
    504: Line8:="I90_SPARE_I504_7(I504.7)        ";
    505: Line8:="I90_SPARE_I505_7(I505.7)        ";
    else
     Line8:=" ";
    END_CASE 
	
  Visibility_1:=TRUE;
   
   CASE IP_Arr_OP90JB[Input_Page_num] OF
	500: Lamp1:=I90_SPARE_I500_0 ;
	501: Lamp1:=I90_CONV1_FWDI501_0 ;
	502: Lamp1:=I90_CONV1_TRK3_CHO_MOD2I502_0 ;
	503: Lamp1:=I90_CONV2_REVI503_0;
	504: Lamp1:=I90_CONV2_TRK3_CHO_MOD1I504_0 ;
	505: Lamp1:=I90_SPARE_I505_0 ;
   ELSE
       Visibility_1:=FALSE;	
   END_CASE
   
   
   Visibility_2:=TRUE;
   
   CASE IP_Arr_OP90JB[Input_Page_num] OF
	500: Lamp2:=I90_HPR1_LOW_LVL_FBI500_1 ;
	501: Lamp2:=I90_VBF1_CONV1_TRK1_OVERFLWI501_1 ;
	502: Lamp2:=I90_SPARE_I502_1 ;
	503: Lamp2:=I90_CONV2_FWDI503_1;
	504: Lamp2:=I90_CONV2_TRK3_CHO_MOD2I504_1 ;
	505: Lamp2:=I90_SPARE_I505_1 ;
   ELSE
       Visibility_2:=FALSE;	
   END_CASE
   
   
    Visibility_3:=TRUE;
   
   CASE IP_Arr_OP90JB[Input_Page_num] OF
	500: Lamp3:=I90_HPR1_SOL_DOOR_SW_FBI500_2 ;
	501: Lamp3:=I90_VBF1_CONV1_TRK2_OVERFLWI501_2 ;
	502: Lamp3:=I90_HPR2_LOW_LVL_FBI502_2 ;
	503: Lamp3:=I90_VBF1_CONV2_TRK1_OVERFLWI503_2;
	504: Lamp3:=I90_VBF1_CONV_TRK_OVERFLW_2I504_2 ;
	505: Lamp3:=I90_SPARE_I505_2 ;
   ELSE
       Visibility_3:=FALSE;	
   END_CASE
   
   
    Visibility_4:=TRUE;
   
   CASE IP_Arr_OP90JB[Input_Page_num] OF
	500: Lamp4:=I90_BOWL1_RDYI500_3 ;
	501: Lamp4:=I90_CONV1_TRK1_CHO_MOD1I501_3 ;
	502: Lamp4:=I90_HPR2_SOL_DOOR_SW_FBI502_3 ;
	503: Lamp4:=I90_VBF1_CONV2_TRK2_OVERFLWI503_3;
	504: Lamp4:=I90_VBF2_CONV_TRK_OVERFLW_2I504_3 ;
	505: Lamp4:=I90_SPARE_I505_3 ;
   ELSE
       Visibility_4:=FALSE;	
   END_CASE
   
   
    Visibility_5:=TRUE;
   
   CASE IP_Arr_OP90JB[Input_Page_num] OF
	500: Lamp5:=I90_BOWL1_LOW_LVLI500_4 ;
	501: Lamp5:=I90_CONV1_TRK1_CHO_MOD2I501_4 ;
	502: Lamp5:=I90_BOWL2_RDYI502_4 ;
	503: Lamp5:=I90_CONV2_TRK1_CHO_MOD1I503_4;
	504: Lamp5:=I90_SPARE_I504_4 ;
	505: Lamp5:=I90_SPARE_I505_4 ;
   ELSE
       Visibility_5:=FALSE;	
   END_CASE
   
   
    Visibility_6:=TRUE;
   
   CASE IP_Arr_OP90JB[Input_Page_num] OF
	500: Lamp6:=I90_BOWL1_OFF_ONI500_5 ;
	501: Lamp6:=I90_CONV1_TRK2_CHO_MOD1I501_5 ;
	502: Lamp6:=I90_BOWL2_LOW_LVLI502_5 ;
	503: Lamp6:=I90_CONV2_TRK1_CHO_MOD2I503_5;
	504: Lamp6:=I90_SPARE_I504_5 ;
	505: Lamp6:=I90_SPARE_I505_5 ;
   ELSE
       Visibility_6:=FALSE;	
   END_CASE
   
   
    Visibility_7:=TRUE;
   
   CASE IP_Arr_OP90JB[Input_Page_num] OF
	500: Lamp7:=I90_HPR1_OFF_ONI500_6 ;
	501: Lamp7:=I90_CONV1_TRK2_CHO_MOD2I501_6 ;
	502: Lamp7:=I90_BOWL2_OFF_ONI502_6 ;
	503: Lamp7:=I90_CONV2_TRK2_CHO_MOD1I503_6;
	504: Lamp7:=I90_SPARE_I504_6 ;
	505: Lamp7:=I90_SPARE_I505_6 ;
   ELSE
       Visibility_7:=FALSE;	
   END_CASE
   
   
    Visibility_8:=TRUE;
   
   CASE IP_Arr_OP90JB[Input_Page_num] OF
	500: Lamp8:=I90_CONV1_REVI500_7 ;
	501: Lamp8:=I90_CONV1_TRK3_CHO_MOD1I501_7 ;
	502: Lamp8:=I90_HPR2_OFF_ONI502_7 ;
	503: Lamp8:=I90_CONV2_TRK2_CHO_MOD2I503_7;
	504: Lamp8:=I90_SPARE_I504_7 ;
	505: Lamp8:=I90_SPARE_I505_7 ;
   ELSE
       Visibility_8:=FALSE;	
   END_CASE
	
    CASE OP_Arr_OP90[Output_Page_num] OF
    500: OLine1:=" O90_HPR1_ENABLE(Q500.0)  ";
    501: OLine1:=" O90_HPR2_ENABLE(Q501.0)  ";
    502: OLine1:=" O90_SPARE_Q502_0(Q502.0) ";
    503: OLine1:=" O90_SPARE_Q503_0(Q503.0) ";
    else
     OLine1:=" ";
    end_case 
    
    CASE OP_Arr_OP90[Output_Page_num] OF
    500: OLine2:="O90_BOWL1_ENABLE(Q500.1)";
    501: OLine2:="O90_BOWL2_ENABLE(Q501.1)";
    502: OLine2:="O90_SPARE_Q502_1(Q502.1)";
    503: OLine2:="O90_SPARE_Q503_1(Q503.1)";
    else
     OLine2:=" ";
    end_case 
    
    CASE OP_Arr_OP90[Output_Page_num] OF
    500: OLine3:="O90_HPR1_TWR_LMP_RED(Q500.2)";
    501: OLine3:="O90_HPR2_TWR_LMP_RED(Q501.2)";
    502: OLine3:="O90_SPARE_Q502_2(Q502.2)    ";
    503: OLine3:="O90_SPARE_Q503_2(Q503.2)    ";
    else
     OLine3:=" ";
    end_case 
    
    CASE OP_Arr_OP90[Output_Page_num] OF
    500: OLine4:="O90_HPR1_TWR_LMP_GREEN(Q500.3)";
    501: OLine4:="O90_HPR2_TWR_LMP_GREEN(Q501.3)";
    502: OLine4:="O90_SPARE_Q502_3(Q502.3)      ";
    503: OLine4:="O90_SPARE_Q503_3(Q503.3)      ";
    else
     OLine4:=" ";
    end_case 
    
    CASE OP_Arr_OP90[Output_Page_num] OF
    500: OLine5:="O90_BOWL1_AIR_PURGE1(Q500.4)";
    501: OLine5:="O90_BOWL2_AIR_PURGE1(Q501.4)";
    502: OLine5:="O90_SPARE_Q502_4(Q502.4)    ";
    503: OLine5:="O90_SPARE_Q503_4(Q503.4)    ";
    else
     OLine5:=" ";
    end_case 
    
    CASE OP_Arr_OP90[Output_Page_num] OF
    500: OLine6:="O90_BOWL1_AIR_PURGE2(Q500.5)";
    501: OLine6:="O90_BOWL2_AIR_PURGE2(Q501.5)";
    502: OLine6:="O90_SPARE_Q502_5(Q502.5)    ";
    503: OLine6:="O90_SPARE_Q503_5(Q503.5)    ";
    else
     OLine6:=" ";
    end_case 
    
    CASE OP_Arr_OP90[Output_Page_num] OF
    500: OLine7:="O90_HPR1_DOOR_OPN(Q500.6)";
    501: OLine7:="O90_HPR2_DOOR_OPN(Q501.6)";
    502: OLine7:="O90_SPARE_Q502_6(Q502.6) ";
    503: OLine7:="O90_SPARE_Q503_6(Q503.6) ";
    else
     OLine7:=" ";
    end_case 
    
    CASE OP_Arr_OP90[Output_Page_num] OF
    500: OLine8:="O90_SPARE_Q500_7(Q500.7)";
    501: OLine8:="O90_SPARE_Q501_7(Q501.7)";
    502: OLine8:="O90_SPARE_Q502_7(Q502.7)";
    503: OLine8:="O90_SPARE_Q503_7(Q503.7)";
    else
     OLine8:=" ";
    END_CASE 
    Out_Visibility_1:=TRUE;
    CASE OP_Arr_OP90[Output_Page_num] OF
	500:  Out_Lamp1:=O90_HPR1_ENABLEQ500_0;
	501:  Out_Lamp1:=O90_HPR2_ENABLEQ501_0;
	502:  Out_Lamp1:=O90_SPARE_Q502_0;
	503:  Out_Lamp1:=O90_SPARE_Q503_0;
    ELSE
       Out_Visibility_1:=FALSE;	
    END_CASE
   
    Out_Visibility_2:=TRUE;
   
    CASE OP_Arr_OP90[Output_Page_num] OF
	500:  Out_Lamp2:=O90_BOWL1_ENABLEQ500_1;
	501:  Out_Lamp2:=O90_BOWL2_ENABLEQ501_1;
	502:  Out_Lamp2:=O90_SPARE_Q502_1;
	503:  Out_Lamp2:=O90_SPARE_Q503_1;
    ELSE
       Out_Visibility_2:=FALSE;	
    END_CASE 
   
    Out_Visibility_3:=TRUE;
	
    CASE OP_Arr_OP90[Output_Page_num] OF
	500:  Out_Lamp3:=O90_HPR1_TWR_LMP_REDQ500_2; 
	501:  Out_Lamp3:=O90_HPR2_TWR_LMP_REDQ501_2; 
	502:  Out_Lamp3:=O90_SPARE_Q502_2; 
	503:  Out_Lamp3:=O90_SPARE_Q503_2; 
    ELSE
       Out_Visibility_3:=FALSE;
    END_CASE 
   
    Out_Visibility_4:=TRUE;
   
    CASE OP_Arr_OP90[Output_Page_num] OF
	500:  Out_Lamp4:=O90_HPR1_TWR_LMP_GREENQ500_3; 
	501:  Out_Lamp4:=O90_HPR2_TWR_LMP_GREENQ501_3; 
	502:  Out_Lamp4:=O90_SPARE_Q502_3; 
	503:  Out_Lamp4:=O90_SPARE_Q503_3;  
    ELSE
       Out_Visibility_4:=FALSE;
    END_CASE 
   
    Out_Visibility_5:=TRUE;
	
    CASE OP_Arr_OP90[Output_Page_num] OF
	500:  Out_Lamp5:=O90_BOWL1_AIR_PURGE1Q500_4; 
	501:  Out_Lamp5:=O90_BOWL2_AIR_PURGE1Q501_4; 
	502:  Out_Lamp5:=O90_SPARE_Q502_4; 
	503:  Out_Lamp5:=O90_SPARE_Q503_4; 
   ELSE
       Out_Visibility_5:=FALSE;
   END_CASE 
   
    Out_Visibility_6:=TRUE;
	
   CASE OP_Arr_OP90[Output_Page_num] OF
	500:  Out_Lamp6:=O90_BOWL1_AIR_PURGE2Q500_5; 
	501:  Out_Lamp6:=O90_BOWL2_AIR_PURGE2Q501_5; 
	502:  Out_Lamp6:=O90_SPARE_Q502_5; 
	503:  Out_Lamp6:=O90_SPARE_Q503_5; 
   ELSE           
       Out_Visibility_6:=FALSE;
   END_CASE 
    
	Out_Visibility_7:=TRUE;
	
   CASE OP_Arr_OP90[Output_Page_num] OF
	500:  Out_Lamp7:=O90_HPR1_DOOR_OPNQ500_6; 
	501:  Out_Lamp7:=O90_HPR2_DOOR_OPNQ501_6; 
	502:  Out_Lamp7:=O90_SPARE_Q502_6; 
	503:  Out_Lamp7:=O90_SPARE_Q503_6;  
   ELSE 
       Out_Visibility_7:=FALSE;
   END_CASE 
   
    Out_Visibility_8:=TRUE;
   
   CASE OP_Arr_OP90[Output_Page_num] OF
	500:  Out_Lamp8:=O90_SPARE_Q500_7;  
	501:  Out_Lamp8:=O90_SPARE_Q501_7;  
	502:  Out_Lamp8:=O90_SPARE_Q502_7;  
	503:  Out_Lamp8:=O90_SPARE_Q503_7;   
   ELSE
       Out_Visibility_8:=FALSE;	
   END_CASE
 7:	CASE IP_Arr_OP120_JB[Input_Page_num] OF
    600: Line1:="I120_SPARE_600_0(I600.0)        ";
    601: Line1:="I120_CONV_FWD(I601.0)           ";
    602: Line1:="I120_CONV_TRK3_CHO_MOD2(I602.0) ";
    603: Line1:="I120_SPARE_I603_0(I603.0)       ";
    else
     Line1:=" ";
    end_case 
     
    CASE IP_Arr_OP120_JB[Input_Page_num] OF
    600: Line2:="I120_HPR_LOW_LVL_FB(I600.1)       ";
    601: Line2:="I120_VBF_CONV_TRK1_OVERFLW(I601.1)";
    602: Line2:="I120_VBF_CONV_TRK_OVERFLW2(I602.1)   ";
    603: Line2:="I120_SPARE_I603_1(I603.1)         ";
    else
     Line2:=" ";
    end_case 
     
    CASE IP_Arr_OP120_JB[Input_Page_num] OF
    600: Line3:="I120_HPR_SOL_DOOR_SW_FB(I600.2)   ";
    601: Line3:="I120_VBF_CONV_TRK2_OVERFLW(I601.2)";
    602: Line3:="I120_SPARE_I602_2(I602.2)         ";
    603: Line3:="I120_SPARE_I603_2(I603.2)         ";
    else
     Line3:=" ";
    end_case 
     
    CASE IP_Arr_OP120_JB[Input_Page_num] OF
    600: Line4:="I120_BOWL_RDY(I600.3)          ";
    601: Line4:="I120_CONV_TRK1_CHO_MOD1(I601.3)";
    602: Line4:="I120_SPARE_I602_3(I602.3)      ";
    603: Line4:="I120_SPARE_I603_3(I603.3)      ";
    else
     Line4:=" ";
    end_case 
     
    CASE IP_Arr_OP120_JB[Input_Page_num] OF
    600: Line5:="I120_BOWL_LOW_LVL(I600.4)      ";
    601: Line5:="I120_CONV_TRK1_CHO_MOD2(I601.4)";
    602: Line5:="I120_SPARE_I602_4(I602.4)      ";
    603: Line5:="I120_SPARE_I603_4(I603.4)      ";
    else
     Line5:=" ";
    end_case 
     
    CASE IP_Arr_OP120_JB[Input_Page_num] OF
    600: Line6:="I120_BOWL_OFF_ON(I600.5)       ";
    601: Line6:="I120_CONV_TRK2_CHO_MOD1(I601.5)";
    602: Line6:="I120_SPARE_I602_5(I602.5)      ";
    603: Line6:="I120_SPARE_I603_5(I603.5)      ";
    else
     Line6:=" ";
    end_case 
     
    CASE IP_Arr_OP120_JB[Input_Page_num] OF
    600: Line7:="I120_HPR_OFF_ON(I600.6)        ";
    601: Line7:="I120_CONV_TRK2_CHO_MOD2(I601.6)";
    602: Line7:="I120_SPARE_I602_6(I602.6)      ";
    603: Line7:="I120_SPARE_I603_6(I603.6)      ";
    else
     Line7:=" ";
    end_case 
     
    CASE IP_Arr_OP120_JB[Input_Page_num] OF
    600: Line8:="I120_CONV_REV(I600.7)           ";
    601: Line8:="I120_CONV_TRK3_CHO_MOD1(I601.7) ";
    602: Line8:="I120_SPARE_I602_7(I602.7)       ";
    603: Line8:="I120_SPARE_I603_7(I603.7)       ";
    else
     Line8:=" ";
    END_CASE 
	Visibility_1:=TRUE;
   
   CASE IP_Arr_OP120_JB[Input_Page_num] OF
	600: Lamp1:=I120_SPARE_600_0I600_0 ;
	601: Lamp1:=I120_CONV_FWDI601_0 ;
	602: Lamp1:=I120_CONV_TRK3_CHO_MOD2I602_0 ;
	603: Lamp1:=I120_SPARE_I603_0;
   ELSE
       Visibility_1:=FALSE;	
   END_CASE
   
   
   Visibility_2:=TRUE;
   
   CASE IP_Arr_OP120_JB[Input_Page_num] OF
	600: Lamp2:=I120_HPR_LOW_LVL_FBI600_1 ;
	601: Lamp2:=I120_VBF_CONV_TRK1_OVERFLWI601_1 ;
	602: Lamp2:=I120_VBF_CONV_TRK_OVERFLW2I602_1 ;
	603: Lamp2:=I120_SPARE_I603_1;
   ELSE
       Visibility_2:=FALSE;	
   END_CASE
   
   
    Visibility_3:=TRUE;
   
   CASE IP_Arr_OP120_JB[Input_Page_num] OF
	600: Lamp3:=I120_HPR_SOL_DOOR_SW_FBI600_2 ;
	601: Lamp3:=I120_VBF_CONV_TRK2_OVERFLWI601_2 ;
	602: Lamp3:=I120_SPARE_I602_2 ;
	603: Lamp3:=I120_SPARE_I603_2;
   ELSE
       Visibility_3:=FALSE;	
   END_CASE

    Visibility_4:=TRUE;
   
   CASE IP_Arr_OP120_JB[Input_Page_num] OF
	600: Lamp4:=I120_BOWL_RDYI600_3 ;
	601: Lamp4:=I120_CONV_TRK1_CHO_MOD1I601_3 ;
	602: Lamp4:=I120_SPARE_I602_3 ;
	603: Lamp4:=I120_SPARE_I603_3;
   ELSE
       Visibility_4:=FALSE;	
   END_CASE
   
   
    Visibility_5:=TRUE;
   
   CASE IP_Arr_OP120_JB[Input_Page_num] OF
	600: Lamp5:=I120_BOWL_LOW_LVLI600_4 ;
	601: Lamp5:=I120_CONV_TRK1_CHO_MOD2I601_4 ;
	602: Lamp5:=I120_SPARE_I602_4 ;
	603: Lamp5:=I120_SPARE_I603_4;
   ELSE
       Visibility_5:=FALSE;	
   END_CASE
   
   
    Visibility_6:=TRUE;
   
   CASE IP_Arr_OP120_JB[Input_Page_num] OF
	600: Lamp6:=I120_BOWL_OFF_ONI600_5 ;
	601: Lamp6:=I120_CONV_TRK2_CHO_MOD1I601_5 ;
	602: Lamp6:=I120_SPARE_I602_5 ;
	603: Lamp6:=I120_SPARE_I603_5;
   ELSE
       Visibility_6:=FALSE;	
   END_CASE
   
   
    Visibility_7:=TRUE;
   
   CASE IP_Arr_OP120_JB[Input_Page_num] OF
	600: Lamp7:=I120_HPR_OFF_ONI600_6 ;
	601: Lamp7:=I120_CONV_TRK2_CHO_MOD2I601_6 ;
	602: Lamp7:=I120_SPARE_I602_6 ;
	603: Lamp7:=I120_SPARE_I603_6;
   ELSE
       Visibility_7:=FALSE;	
   END_CASE
   
   
    Visibility_8:=TRUE;
   
   CASE IP_Arr_OP120_JB[Input_Page_num] OF
	600: Lamp8:=I120_CONV_REVI600_7 ;
	601: Lamp8:=I120_CONV_TRK3_CHO_MOD1I601_7 ;
	602: Lamp8:=I120_SPARE_I602_7 ;
	603: Lamp8:=I120_SPARE_I603_7;
   ELSE
       Visibility_8:=FALSE;	
   END_CASE
    
    CASE OP_Arr_OP120[Output_Page_num] OF
    600: OLine1:="O120_HPR_ENABLE(Q600.0)   ";
    601: OLine1:="O120_SPARE_Q601_0(Q601.0) ";
    602: OLine1:="O120_SPARE_Q602_0(Q602.0) ";
    603: OLine1:="O120_SPARE_Q603_0(Q603.0) ";
    else
     OLine1:=" ";
    end_case 
    
    CASE OP_Arr_OP120[Output_Page_num] OF
    600: OLine2:="O120_BOWL_ENABLE(Q600.1) ";
    601: OLine2:="O120_SPARE_Q601_1(Q601.1)";
    602: OLine2:="O120_SPARE_Q602_1(Q602.1)";
    603: OLine2:="O120_SPARE_Q603_1(Q603.1)";
    else
     OLine2:=" ";
    end_case 
    
    CASE OP_Arr_OP120[Output_Page_num] OF
    600: OLine3:="O120_HPR_TWR_LMP_RED(Q600.2)";
    601: OLine3:="O120_SPARE_Q601_2(Q601.2)   ";
    602: OLine3:="O120_SPARE_Q602_2(Q602.2)   ";
    603: OLine3:="O120_SPARE_Q603_2(Q603.2)   ";
    else
     OLine3:=" ";
    end_case 
    
    CASE OP_Arr_OP120[Output_Page_num] OF
    600: OLine4:="O120_HPR_TWR_LMP_GREEN(Q600.3)";
    601: OLine4:="O120_SPARE_Q601.3(Q601.3)     ";
    602: OLine4:="O120_SPARE_Q602.3(Q602.3)     ";
    603: OLine4:="O120_SPARE_Q603.3(Q603.3)     ";
    else
     OLine4:=" ";
    end_case 
    
    CASE OP_Arr_OP120[Output_Page_num] OF
    600: OLine5:="O120_BOWL_AIR_PURGE1(Q600.4)";
    601: OLine5:="O120_SPARE_Q601_4(Q601.4)   ";
    602: OLine5:="O120_SPARE_Q602_4(Q602.4)   ";
    603: OLine5:="O120_SPARE_Q603_4(Q603.4)   ";
    else
     OLine5:=" ";
    end_case 
    
    CASE OP_Arr_OP120[Output_Page_num] OF
    600: OLine6:="O120_BOWL_AIR_PURGE2(Q600.5)";
    601: OLine6:="O120_SPARE_Q601_5(Q601.5)   ";
    602: OLine6:="O120_SPARE_Q602_5(Q602.5)   ";
    603: OLine6:="O120_SPARE_Q603_5(Q603.5)   ";
    else
     OLine6:=" ";
    end_case 
    
    CASE OP_Arr_OP120[Output_Page_num] OF
    600: OLine7:="O120_HPR_DOOR_OPN(Q600.6)";
    601: OLine7:="O120_SPARE_Q601_6(Q601.6)";
    602: OLine7:="O120_SPARE_Q602_6(Q602.6)";
    603: OLine7:="O120_SPARE_Q603_6(Q603.6)";
    else
     OLine7:=" ";
    end_case 
    
    CASE OP_Arr_OP120[Output_Page_num] OF
    600: OLine8:="O120_SPARE_Q600_7(Q600.7)";
    601: OLine8:="O120_SPARE_Q601_7(Q601.7)";
    602: OLine8:="O120_SPARE_Q602_7(Q602.7)";
    603: OLine8:="O120_SPARE_Q603_7(Q603.7)";
    else
     OLine8:=" ";
    END_CASE 
	   Out_Visibility_1:=TRUE;
   
   CASE OP_Arr_OP120[Output_Page_num] OF
	600:  Out_Lamp1:=O120_HPR_ENABLEQ600_0;
	601:  Out_Lamp1:=O120_SPARE_Q601_0;
	602:  Out_Lamp1:=O120_SPARE_Q602_0;
	603:  Out_Lamp1:=O120_SPARE_Q603_0;
   ELSE
       Out_Visibility_1:=FALSE;	
   END_CASE
   
    Out_Visibility_2:=TRUE;
   
   CASE OP_Arr_OP120[Output_Page_num] OF
	600:  Out_Lamp2:=O120_BOWL_ENABLEQ600_1;
	601:  Out_Lamp2:=O120_SPARE_Q601_1;
	602:  Out_Lamp2:=O120_SPARE_Q602_1;
	603:  Out_Lamp2:=O120_SPARE_Q603_1;
   ELSE
       Out_Visibility_2:=FALSE;	
   END_CASE 
   
    Out_Visibility_3:=TRUE;
	
   CASE OP_Arr_OP10A[Output_Page_num] OF
	600:  Out_Lamp3:=O120_HPR_TWR_LMP_REDQ600_2; 
	601:  Out_Lamp3:=O120_SPARE_Q601_2; 
	602:  Out_Lamp3:=O120_SPARE_Q602_2; 
	603:  Out_Lamp3:=O120_SPARE_Q603_2; 
   ELSE
       Out_Visibility_3:=FALSE;
   END_CASE 
   
    Out_Visibility_4:=TRUE;
   
   CASE OP_Arr_OP120[Output_Page_num] OF
	700:  Out_Lamp4:=O120_HPR_TWR_LMP_GREENQ600_3; 
	701:  Out_Lamp4:=O120_SPARE_Q601_3; 
	702:  Out_Lamp4:=O120_SPARE_Q602_3; 
	703:  Out_Lamp4:=O120_SPARE_Q603_3; 
   ELSE
       Out_Visibility_4:=FALSE;
   END_CASE 
   
    Out_Visibility_5:=TRUE;
	
    CASE OP_Arr_OP120[Output_Page_num] OF
	600:  Out_Lamp5:=O120_BOWL_AIR_PURGE1Q600_4; 
	601:  Out_Lamp5:=O120_SPARE_Q601_4; 
	602:  Out_Lamp5:=O120_SPARE_Q602_4; 
	603:  Out_Lamp5:=O120_SPARE_Q603_4; 
   ELSE
       Out_Visibility_5:=FALSE;
   END_CASE 
   
    Out_Visibility_6:=TRUE;
	
   CASE OP_Arr_OP120[Output_Page_num] OF
	600:  Out_Lamp6:=O120_BOWL_AIR_PURGE2Q600_5; 
	601:  Out_Lamp6:=O120_SPARE_Q601_5; 
	602:  Out_Lamp6:=O120_SPARE_Q602_5; 
	603:  Out_Lamp6:=O120_SPARE_Q603_5; 
   ELSE           
       Out_Visibility_6:=FALSE;
   END_CASE 
    
	Out_Visibility_7:=TRUE;
	
   CASE OP_Arr_OP120[Output_Page_num] OF
	600:  Out_Lamp7:=O120_HPR_DOOR_OPNQ600_6; 
	601:  Out_Lamp7:=O120_SPARE_Q601_6; 
	602:  Out_Lamp7:=O120_SPARE_Q602_6; 
	603:  Out_Lamp7:=O120_SPARE_Q603_6; 
   ELSE 
       Out_Visibility_7:=FALSE;
   END_CASE 
   
    Out_Visibility_8:=TRUE;
   
   CASE OP_Arr_OP120[Output_Page_num] OF
	600:  Out_Lamp8:=O120_SPARE_Q600_7;  
	601:  Out_Lamp8:=O120_SPARE_Q601_7;  
	602:  Out_Lamp8:=O120_SPARE_Q602_7;  
	603:  Out_Lamp8:=O120_SPARE_Q603_7;  
   ELSE
       Out_Visibility_8:=FALSE;	
   END_CASE
	
 8: CASE Safety_IP[Input_Page_num] OF
    400: Line1:="IS90_DOORSW_SET1_CH1(IS400.0)";
    401: Line1:="IS90_DOORSW_SET5_CH1(IS401.0)";
    402: Line1:="IS90_ESTOP_CONT_EDM(IS402.0) ";
    700: Line1:="IS160_ESTOP_CONT_EDM(IS700.0)";
    else
     Line1:=" ";
    END_CASE 
    
    CASE Safety_IP[Input_Page_num] OF
    400: Line2:="IS90_DOORSW_SET2_CH1(IS400.1)";
    401: Line2:="IS90_DOORSW_SET6_CH1(IS401.1)";
    402: Line2:="IS90_DOOR_CONT_EDM(IS402.1)  ";
    700: Line2:="IS160_DOOR_CONT_EDM(IS700.1) ";
    else
     Line2:=" ";
    end_case 
    
    
    CASE Safety_IP[Input_Page_num] OF
    400: Line3:="IS90_DOORSW_SET3_CH1(IS400.2)";
    401: Line3:="IS90_LHS_ESTOP_CH1(IS401.2)  ";
    402: Line3:="IS90_RESET_IS402_2(IS402.2)  ";
    700: Line3:="IS160_SPARE_IS700_2(IS700.2) ";
    else
     Line3:=" ";
    end_case 
    
    
    CASE Safety_IP[Input_Page_num] OF
    400: Line4:="IS90_DOORSW_SET4_CH1(IS400.3)";
    401: Line4:="IS90_RHS_ESTOP_CH1(IS401.3)  ";
    402: Line4:="IS90_SPARE_IS402_3(IS402.3)  ";
    700: Line4:="IS160_SPARE_IS700_3(IS700.3) ";
    else
     Line4:=" ";
    end_case 
    
    CASE Safety_IP[Input_Page_num] OF
    400: Line5:="IS90_DOORSW_SET1_CH2(IS400.4)";
    401: Line5:="IS90_DOORSW_SET5_CH2(IS401.4)";
    402: Line5:="IS90_SPARE_IS402_4(IS402.4)  ";
    700: Line5:="IS160_SPARE_IS700_4(IS700.4) ";
    else
     Line5:=" ";
    end_case 
    
    CASE Safety_IP[Input_Page_num] OF
    400: Line6:="IS90_DOORSW_SET2_CH2(IS400.5)";
    401: Line6:="IS90_DOORSW_SET6_CH2(IS401.5)";
    402: Line6:="IS90_SPARE_IS402_5(IS402.5)  ";
    700: Line6:="IS160_SPARE_IS700_5(IS700.5) ";
    else
     Line6:=" ";
    end_case 
    
    CASE Safety_IP[Input_Page_num] OF
    400: Line7:="IS90_DOORSW_SET3_CH2(IS400.6)";
    401: Line7:="IS90_LHS_ESTOP_CH2(IS401.6)  ";
    402: Line7:="IS90_SPARE_IS402_6(IS402.6)  ";
    700: Line7:="IS160_SPARE_IS700_6(IS700.6) ";
    else
     Line7:=" ";
    end_case 
    
    CASE Safety_IP[Input_Page_num] OF
    400: Line8:="IS90_DOORSW_SET4_CH2(IS400.7)";
    401: Line8:="IS90_RHS_ESTOP_CH2(IS401.7)  ";
    402: Line8:="IS90_SPARE_IS402_7(IS402.7)  ";
    700: Line8:="IS160_SPARE_IS700_7(IS700.7) ";
    else
     Line8:=" ";
    END_CASE 
	   Visibility_1:=TRUE;
   
   CASE Safety_IP[Input_Page_num] OF
	400: Lamp1:=IS90_DOORSW_SET1_CH1_IS400_0 ;
	401: Lamp1:=IS90_DOORSW_SET5_CH1_IS401_0 ;
	402: Lamp1:=IS90_ESTOP_CONT_EDM_IS402_0 ;
	700: Lamp1:=IS160_ESTOP_CONT_EDM_IS700_0;
   ELSE
       Visibility_1:=FALSE;	
   END_CASE
   
   
   Visibility_2:=TRUE;
   
   CASE Safety_IP[Input_Page_num]OF
	400: Lamp2:=IS90_DOORSW_SET2_CH1_IS400_1 ;
	401: Lamp2:=IS90_DOORSW_SET6_CH1_IS401_1 ;
	402: Lamp2:=IS90_DOOR_CONT_EDM_IS402_1 ;
	700: Lamp2:=IS160_DOOR_CONT_EDM_IS700_1;
   ELSE
       Visibility_2:=FALSE;	
   END_CASE
   
   
    Visibility_3:=TRUE;
   
   CASE Safety_IP[Input_Page_num] OF
	400: Lamp3:=IS90_DOORSW_SET3_CH1_IS400_2 ;
	401: Lamp3:=IS90_LHS_ESTOP_CH1_IS401_2 ;
	402: Lamp3:=IS90_RESET_IS402_2 ;
	700: Lamp3:=IS160_SPARE_IS700_2;
   ELSE
       Visibility_3:=FALSE;	
   END_CASE
   
   
    Visibility_4:=TRUE;
   
   CASE Safety_IP[Input_Page_num] OF
	400: Lamp4:=IS90_DOORSW_SET4_CH1_IS400_3 ;
	401: Lamp4:=IS90_RHS_ESTOP_CH1_IS401_3 ;
	402: Lamp4:=IS90_SPARE_IS402_3 ;
	700: Lamp4:=IS160_SPARE_IS700_3;
   ELSE
       Visibility_4:=FALSE;	
   END_CASE
   
   
    Visibility_5:=TRUE;
   
   CASE Safety_IP[Input_Page_num] OF
	400: Lamp5:=IS90_DOORSW_SET1_CH2_IS400_4 ;
	401: Lamp5:=IS90_DOORSW_SET5_CH2_IS401_4 ;
	402: Lamp5:=IS90_SPARE_IS402_4 ;
	700: Lamp5:=IS160_SPARE_IS700_4;
   ELSE
       Visibility_5:=FALSE;	
   END_CASE
   
   
    Visibility_6:=TRUE;
   
   CASE Safety_IP[Input_Page_num] OF
	400: Lamp6:=IS90_DOORSW_SET2_CH2_IS400_5 ;
	401: Lamp6:=IS90_DOORSW_SET6_CH2_IS401_5 ;
	402: Lamp6:=IS90_SPARE_IS402_5 ;
	700: Lamp6:=IS160_SPARE_IS700_5;
   ELSE
       Visibility_6:=FALSE;	
   END_CASE
   
   
    Visibility_7:=TRUE;
   
   CASE Safety_IP[Input_Page_num] OF
	400: Lamp7:=IS90_DOORSW_SET3_CH2_IS400_6 ;
	401: Lamp7:=IS90_LHS_ESTOP_CH2_IS401_6 ;
	402: Lamp7:=IS90_SPARE_IS402_6 ;
	700: Lamp7:=IS160_SPARE_IS700_6;
   ELSE
       Visibility_7:=FALSE;	
   END_CASE
   
   
    Visibility_8:=TRUE;
   
   CASE Safety_IP[Input_Page_num] OF
	400: Lamp8:=IS90_DOORSW_SET4_CH2_IS400_7 ;
	401: Lamp8:=IS90_RHS_ESTOP_CH2_IS401_7 ;
	402: Lamp8:=IS90_SPARE_IS402_7 ;
	700: Lamp8:=IS160_SPARE_IS700_7;
   ELSE
       Visibility_8:=FALSE;	
   END_CASE

	CASE Safety_OP[Output_Page_num] OF
    400: OLine1:="OS90_ESTOP_CH1(QS400.0) ";
    700: OLine1:="OS160_ESTOP_CH1(QS700.0)";
    else
     OLine1:=" ";
    end_case 
    
    CASE Safety_OP[Output_Page_num] OF
    400: OLine2:="OS90_ESTOP_CH2(QS400.1) ";
    700: OLine2:="OS160_ESTOP_CH2(QS700.1)";
    else
     OLine2:=" ";
    end_case 
    
    CASE Safety_OP[Output_Page_num] OF
    400: OLine3:="OS90_DOORCH1(QS400.2)  ";
    700: OLine3:="OS160_DOORCH1(QS700.2) ";
    else
     OLine3:=" ";
    end_case 
    
    CASE Safety_OP[Output_Page_num] OF
    400: OLine4:="OS90_DOORCH2(QS400.3) ";
    700: OLine4:="OS160_DOORCH2(QS700.3)";
    else
     OLine4:=" ";
    END_CASE
	
	   Out_Visibility_1:=TRUE;
   
   CASE Safety_OP[Output_Page_num] OF
	400:  Out_Lamp1:=OS90_ESTOP_CH1_QS400_0;
	700:  Out_Lamp1:=OS160_ESTOP_CH1_QS700_0;
   ELSE
       Out_Visibility_1:=FALSE;	
   END_CASE
   
    Out_Visibility_2:=TRUE;
   
   CASE Safety_OP[Output_Page_num] OF
	400:  Out_Lamp2:=OS90_ESTOP_CH2_QS400_1;
	700:  Out_Lamp2:=OS160_ESTOP_CH2_QS700_1;
   ELSE
       Out_Visibility_2:=FALSE;	
   END_CASE 
   
    Out_Visibility_3:=TRUE;
	
   CASE Safety_OP[Output_Page_num] OF
	400:  Out_Lamp3:=OS90_DOORCH1_QS400_2; 
	700:  Out_Lamp3:=OS160_DOORCH1_QS700_2; 
   ELSE
       Out_Visibility_3:=FALSE;
   END_CASE 
   
    Out_Visibility_4:=TRUE;
   
    CASE Safety_OP[Output_Page_num] OF
	400:  Out_Lamp4:=OS90_DOORCH2_QS400_3; 
	700:  Out_Lamp4:=OS160_DOORCH2_QS700_3; 
    ELSE
	   Out_Visibility_4:=FALSE;
    END_CASE 
	   
    
    Out_Visibility_5:=FALSE; 
    Out_Visibility_6:=FALSE;
    Out_Visibility_7:=FALSE;
    Out_Visibility_8:=FALSE;
   
END_CASE	 

IF panel_num = 1 THEN
i:= IP_Arr_OP10P[Input_Page_num];
j:= OP_Arr_OP10P[Output_Page_num];	
 IF Input_Page_num >= 26 THEN
	Input_Page_num:=0;
 END_IF
 IF Output_Page_num >= 21 THEN
	Output_Page_num:=0;
 END_IF	
END_IF

IF panel_num = 2 THEN
i:= IP_Arr_OP90P[Input_Page_num];
j:= OP_Arr_OP90P[Output_Page_num];	
 IF Input_Page_num >= 12 THEN
	Input_Page_num:=0;
 END_IF
 IF Output_Page_num >= 10 THEN
	Output_Page_num:=0;
 END_IF	
END_IF

IF panel_num = 3 THEN
i:= IP_Arr_OP160P[Input_Page_num];
j:= OP_Arr_OP160P[Output_Page_num];	
 IF Input_Page_num >= 9 THEN
	Input_Page_num:=0;
 END_IF
 IF Output_Page_num >= 9 THEN
	Output_Page_num:=0;
 END_IF	
END_IF

IF panel_num = 4 THEN
i:= IP_Arr_OP10A[Input_Page_num];
j:= OP_Arr_OP10A[Output_Page_num];	
 IF Input_Page_num >= 4 THEN
	Input_Page_num:=0;
 END_IF
 IF Output_Page_num >= 4 THEN
	Output_Page_num:=0;
 END_IF	
END_IF

IF panel_num = 5 THEN
i:= IP_Arr_OP10B[Input_Page_num];
j:= OP_Arr_OP10B_JB[Output_Page_num];	
 IF Input_Page_num >= 4 THEN
	Input_Page_num:=0;
 END_IF
 IF Output_Page_num >= 4 THEN
	Output_Page_num:=0;
 END_IF	
END_IF

IF panel_num = 6 THEN
i:= IP_Arr_OP90JB[Input_Page_num];
j:= OP_Arr_OP90[Output_Page_num];	
 IF Input_Page_num >= 6 THEN
	Input_Page_num:=0;
 END_IF
 IF Output_Page_num >= 4 THEN
	Output_Page_num:=0;
 END_IF	
END_IF

IF panel_num = 7 THEN
i:= IP_Arr_OP120_JB[Input_Page_num];
j:= OP_Arr_OP120[Output_Page_num];	
 IF Input_Page_num >= 4 THEN
	Input_Page_num:=0;
 END_IF
 IF Output_Page_num >= 4 THEN
	Output_Page_num:=0;
 END_IF	
END_IF

IF panel_num = 8 THEN
 OLine5:=" ";
 OLine6:=" ";
 OLine7:=" ";
 OLine8:=" ";	
 i:= Safety_IP[Input_Page_num];
 j:= Safety_OP[Output_Page_num];	
  IF Input_Page_num >= 4 THEN
 	Input_Page_num:=0;
  END_IF
  IF Output_Page_num >= 2 THEN
 	Output_Page_num:=0;
  END_IF	
END_IF

END_PROGRAM

(* stored: Version 1.1.0.1, ProductVersion 3.1.4024.11
   POU IO_Dig: Id {372675bb-47f2-47b8-be5b-a3062772c492}, SpecialFunc None *)
